// LS Electric XG5000 project: 9_3_시험문제 1번 연습
// PLC LSPLC
// module base 0 slot 0: 입출력 모듈:XBC-DR14E (DC 24V 입력 8점, 릴레이 출력 6점)

PROGRAM NewProgram (task: 스캔 프로그램)

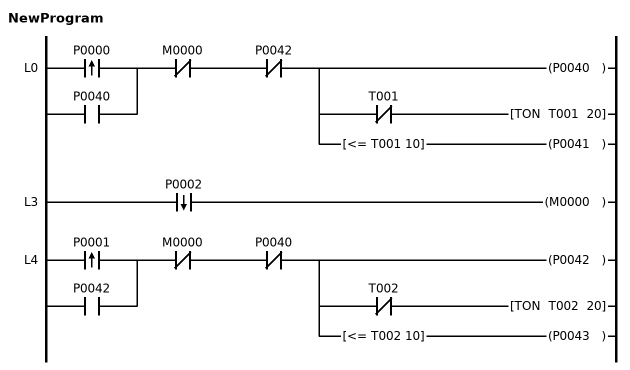
; L0
LOADP     P0000
OR        P0040
AND NOT   M0000
AND NOT   P0042
OUT       P0040
MPUSH
AND NOT   T001
TON       T001 20
MPOP
AND<=     T001 10
OUT       P0041
; L3
LOADN     P0002
OUT       M0000
; L4
LOADP     P0001
OR        P0042
AND NOT   M0000
AND NOT   P0040
OUT       P0042
MPUSH
AND NOT   T002
TON       T002 20
MPOP
AND<=     T002 10
OUT       P0043